// TIA Portal V18 export
DATA_BLOCK "MotorControl"   // DB3100
{ S7_Optimized_Access := 'TRUE' }
VERSION : 0.1
// stored: AutoNumber false, DBAccessibleFromOPCUA true, DBAccessibleFromWebserver true, IsOnlyStoredInLoadMemory false, IsRetainMemResEnabled false, IsWriteProtectedInAS false, MemoryReserve 100
   VAR
      Dev : Array[1..20] of "Motor_Control";
   END_VAR
BEGIN
END_DATA_BLOCK
